Staubli VAL3: AfterTraj.pgx

public program AfterTraj(num x_nWorkplaceIn, num x_nTrajIndex)
begin
  //参数：x_nWorkplaceIn 工位序号，传入的参数是 DataBase:nWorkPlaceIndex
  //参数：x_nTrajIndex 路径序号，传入的参数是TxtFile:nReadTrajIndex
  //引用位置:Motion:Move.pgx
  //功能：用在完成离开点之后
  //备注：添加动作需要waitendmove()
  //

  //
  //    if bDebug
  //    popUpMsg("AfterTraj")
  //    logMsg("AfterTraj")
  //
  //
  //    endIf






















end
